(* CODESYS project HomePLC_LinkManager.library
   Company: Tom Oyen
   Description: Link manager
   Version: 1.0
   Placeholder: HomePLC Link Manager
   Author: Tom Oyen
   Title: HomePLC Link Manager

Project tree, tasks and I/O mapping:
  libraries: Tc2_Standard, * (Beckhoff Automation GmbH); Tc2_System, * (Beckhoff Automation GmbH); Tc3_Module, * (Beckhoff Automation GmbH); HomePLC Logging, * (Tom Oyen); HomePLC DIO, * (Tom Oyen)
  POUs/
    IO group/
      DUTs/
        data type E_DIGroupMode
      function block FB_DIGroup [ST]: AddInput, Execute, GetCommand, GetInput, Mode
      function block FB_DOGroup [ST]: AddOutput, Execute, GetOutput, SetCommand
      function block FB_IOGroup [ST]: FB_init, Count
      interface I_DIGroup: AddInput, GetCommand, GetInput, Count, Mode
      interface I_DOGroup: AddOutput, GetOutput, SetCommand, Count
    Link/
      DUTs/
        data type ST_CommandTranslation
      function block FB_Link [ST]: Execute, FB_init, ExcludeFromOverview, InputGroup, OutputGroup, OutputReaction
      interface I_Link: ExcludeFromOverview, InputGroup, OutputGroup, OutputReaction
    function block FB_LinkManager [ST]: CommitLink, Execute, GetLink, Link
    interface I_LinkManager: CommitLink, Link
  Project Information/
    function F_GetCompany [ST]
    function F_GetTitle [ST]
    function F_GetVersion [ST]
  Version/
    global variables Global_Version
*)

// POUs/IO group/DUTs/E_DIGroupMode
{attribute 'qualified_only'}
{attribute 'strict'}
// Mode of combining digital input commands
TYPE E_DIGroupMode :
(
	ModeAND := 0,		// All inputs need to be used to issue the command
	ModeOR	:= 1		// One input is sufficient to issue a command
);
END_TYPE

// POUs/Link/DUTs/ST_CommandTranslation
// Translate input commands to output commands
TYPE ST_CommandTranslation :
STRUCT
	OnShortPress	: E_DOCommand := E_DOCommand.None;	// Output command when input command is short press
	OnLongPress		: E_DOCommand := E_DOCommand.None;	// Output command when input command is long press
	OnDoublePress	: E_DOCommand := E_DOCommand.None;	// Output command when input command is double press
	OnHold			: E_DOCommand := E_DOCommand.None;	// Output command when input command is hold
END_STRUCT
END_TYPE

// Version/Global_Version
{attribute 'TcGenerated'}
{attribute 'no-analysis'}
{attribute 'linkalways'}
// This function has been automatically generated from the project information.
VAR_GLOBAL CONSTANT
	{attribute 'const_non_replaced'}
	stLibVersion_HomePLC_Link_Manager : ST_LibVersion := (iMajor := 1, iMinor := 0, iBuild := 0, iRevision := 0, nFlags := 0, sVersion := '1.0');
END_VAR

// POUs/IO group/FB_DIGroup
// Digital input group
FUNCTION_BLOCK FB_DIGroup EXTENDS FB_IOGroup IMPLEMENTS I_DIGroup
VAR
	aIn				: ARRAY [0..nMaxSize - 1] OF I_DigitalIn;	// Array of interfaces of digital inputs
	eMode			: E_DIGroupMode := E_DIGroupMode.ModeOR;	// Command mode of inputs in group (default = OR)
END_VAR

// Add input to group
METHOD AddInput
VAR_INPUT
	IDI			: I_DigitalIn;
END_VAR
IF nSize < nMaxSize THEN
	aIn[nSize] := IDI;
	nSize := nSize + 1;
END_IF
END_METHOD

// Runs the execute method of all digital input FBs in the group
METHOD Execute
VAR
	i		: INT;
END_VAR
FOR i := 0 TO nSize - 1 DO
	aIn[i].Execute();
END_FOR
END_METHOD

// Determine the command from the inputs in the group
METHOD GetCommand : E_DICommand
VAR
	i				: INT;
	nActive			: INT;
	eCommand		: E_DICommand;
	sTemp			: STRING;
END_VAR
VAR_INST
	eState			: E_DIState;
END_VAR
// Check at least one input is available
IF nSize > 0 THEN
	CASE eMode OF
	E_DIGroupMode.ModeOR:
		// Get command
		eCommand := E_DICommand.None;
		
		FOR i := 0 TO nSize - 1 DO
			// Find first command different from None
			IF aIn[i].Command <> E_DICommand.None THEN
				IF eCommand = E_DICommand.None THEN
					eCommand := aIn[i].Command;
					
					sTemp := 'OR command ';
					sTemp := CONCAT(sTemp, TO_STRING(eCommand));
					fbLogger.AddDebug(sTemp);
				END_IF
			END_IF
		END_FOR
		
		// Issue command
		GetCommand := eCommand;
		
	E_DIGroupMode.ModeAND:
		// Check states
		// Multiple buttons must have been active at the same time with the same state
		nActive := 0;
		FOR i := 0 TO nSize - 1 DO
			IF aIn[i].State <> E_DIState.Idle THEN
				IF eState = E_DIState.Idle THEN
					eState := aIn[i].State;
				END_IF
				IF aIn[i].State = eState THEN
					nActive := nActive + 1;
				END_IF
			END_IF
		END_FOR
		
		// Reset if all inactive
		IF nActive = 0 THEN
			eState := E_DIState.Idle;
		END_IF
		
		// Get command
		eCommand := E_DICommand.None;
		FOR i := 0 TO nSize - 1 DO
			// Find first command different from None
			IF aIn[i].Command <> E_DICommand.None THEN
				IF eCommand = E_DICommand.None THEN
					eCommand := aIn[i].Command;
				END_IF
			END_IF
		END_FOR
		
		IF eCommand <> E_DICommand.None THEN
			// All commands need to be the same
			// Assume command matches detected states
			IF nActive = nSize THEN
				GetCommand := eCommand;
				
				sTemp := 'AND command ';
				sTemp := CONCAT(sTemp, TO_STRING(eCommand));
				sTemp := CONCAT(sTemp, ' by ');
				sTemp := CONCAT(sTemp, INT_TO_STRING(nActive));
				sTemp := CONCAT(sTemp, ' inputs');
				fbLogger.AddDebug(sTemp);
			END_IF
		ELSE
			GetCommand := E_DICommand.None;
		END_IF
	END_CASE
ELSE
	GetCommand := E_DICommand.None;
END_IF
END_METHOD

// Get a specific input from the group
METHOD GetInput : I_DigitalIn
VAR_INPUT
	nInputIndex		: INT;		// Input index
END_VAR
GetInput := aIn[nInputIndex];
END_METHOD

// Set input group mode (default OR)
PROPERTY Mode : E_DIGroupMode
SET
eMode := Mode;
END_SET
END_PROPERTY

END_FUNCTION_BLOCK

// POUs/IO group/FB_IOGroup
{attribute 'reflection'} 
FUNCTION_BLOCK FB_IOGroup
VAR
	nSize			: INT;			// Number of IOs in this group
	
	fbLogger		: class_Tc3EventLogger;
	
	// Use attributes to copy instance name to sName
	{attribute 'instance-path'} 
    {attribute 'noinit'} 
    sName			: STRING; 		// Instance name
END_VAR
VAR CONSTANT
	nMaxSize		: INT := 100;	// Maximum number of IOs in a group
END_VAR

METHOD FB_init : BOOL
VAR_INPUT
	bInitRetains : BOOL; // if TRUE, the retain variables are initialized (warm start / cold start)
	bInCopyCode : BOOL;  // if TRUE, the instance afterwards gets moved into the copy code (online change)
END_VAR
fbLogger.Init(sSource := sName, bEnableVerbose := FALSE);
END_METHOD

// Gets the total number of IOs in the group
PROPERTY Count : INT
GET
Count := nSize;
END_GET
END_PROPERTY

END_FUNCTION_BLOCK

// POUs/IO group/I_DIGroup
INTERFACE I_DIGroup

// Add input to group
METHOD AddInput
VAR_INPUT
	IDI			: I_DigitalIn;		// Digital input
END_VAR
END_METHOD

// Determine the command from the inputs in the group
METHOD GetCommand : E_DICommand
END_METHOD

// Get a specific input from the group
METHOD GetInput : I_DigitalIn
VAR_INPUT
	nInputIndex		: INT;		// Input index
END_VAR
END_METHOD

// Gets the total number of IOs in the group
PROPERTY Count : INT
GET
END_GET
END_PROPERTY

// Set input group mode (default OR)
PROPERTY Mode : E_DIGroupMode
SET
END_SET
END_PROPERTY

END_INTERFACE

// POUs/IO group/FB_DOGroup
// Digital output group
FUNCTION_BLOCK FB_DOGroup EXTENDS FB_IOGroup IMPLEMENTS I_DOGroup
VAR
	aOut		: ARRAY [0..nMaxSize - 1] OF I_DigitalOut;		// Array of interfaces to digital outputs
END_VAR

// Add output to group
METHOD AddOutput
VAR_INPUT
	IDO			: I_DigitalOut;
END_VAR
IF nSize < nMaxSize THEN
	aOut[nSize] := IDO;
	nSize := nSize + 1;
END_IF
END_METHOD

// Runs the execute method of all digital output FBs in the group
METHOD Execute
VAR
	i		: INT;
END_VAR
FOR i := 0 TO nSize - 1 DO
	aOut[i].Execute();
END_FOR
END_METHOD

// Get a specific output from the group
METHOD GetOutput : I_DigitalOut
VAR_INPUT
	nOutputIndex		: INT;		// Output index
END_VAR
GetOutput := aOut[nOutputIndex];
END_METHOD

// Set the command to the outputs in the group
METHOD SetCommand
VAR_INPUT
	eCommand	: E_DOCommand;
END_VAR
VAR
	i			: INT;
END_VAR
FOR i := 0 TO nSize - 1 DO
	IF aOut[i].Command = E_DOCommand.None THEN
		// No command yet, set new command
		aOut[i].SetCommand(eCommand);
	ELSE
		// A command was already issued
		// Do nothing
	END_IF
END_FOR
END_METHOD

END_FUNCTION_BLOCK

// POUs/IO group/I_DOGroup
INTERFACE I_DOGroup

// Add output to group
METHOD AddOutput
VAR_INPUT
	IDO			: I_DigitalOut;		// Digital output
END_VAR
END_METHOD

// Get a specific output from the group
METHOD GetOutput : I_DigitalOut
VAR_INPUT
	nOutputIndex		: INT;		// Output index
END_VAR
END_METHOD

// Set the command to the outputs in the group
METHOD SetCommand
VAR_INPUT
	eCommand	: E_DOCommand;
END_VAR
END_METHOD

// Gets the total number of IOs in the group
PROPERTY Count : INT
GET
END_GET
END_PROPERTY

END_INTERFACE

// POUs/Link/FB_Link
// Link between an input and an output group
FUNCTION_BLOCK FB_Link IMPLEMENTS I_Link
VAR
	IInputGroup				: I_DIGroup;				// Input group interface
	IOutputGroup			: I_DOGroup;				// Output group interface
	
	fbInputGroup			: FB_DIGroup;				// Input group FB, in case interface is not set to an FB
	fbOutputGroup			: FB_DOGroup;				// Output group FB, in case interface is not set to an FB
	
	stCommandTranslation	: ST_CommandTranslation;	// Input command to output command translation
	bExcludeFromOverview	: BOOL;						// Set to true to exclude this link from the links overview
END_VAR

// Execute input group, get its command and then execute the output group with that command
METHOD Execute
// Get input command and translate it to an output command
CASE IInputGroup.GetCommand() OF
	E_DICommand.None:
		IOutputGroup.SetCommand(E_DOCommand.None);
	E_DICommand.ShortPress:
		IOutputGroup.SetCommand(stCommandTranslation.OnShortPress);
	E_DICommand.DoublePress:
		IOutputGroup.SetCommand(stCommandTranslation.OnDoublePress);
	E_DICommand.LongPress:
		IOutputGroup.SetCommand(stCommandTranslation.OnLongPress);
	E_DICommand.Hold:
		IOutputGroup.SetCommand(stCommandTranslation.OnHold);
END_CASE
END_METHOD

METHOD FB_init : BOOL
VAR_INPUT
	bInitRetains : BOOL; // if TRUE, the retain variables are initialized (warm start / cold start)
	bInCopyCode : BOOL;  // if TRUE, the instance afterwards gets moved into the copy code (online change)
END_VAR
// Initialize interfaces with local FBs, can be replaced afterwards if needed
IInputGroup := fbInputGroup;
IOutputGroup := fbOutputGroup;
END_METHOD

// Get/set if the link needs to be excluded from the links overview
PROPERTY ExcludeFromOverview : BOOL
GET
ExcludeFromOverview := bExcludeFromOverview;
END_GET
SET
bExcludeFromOverview := ExcludeFromOverview;
END_SET
END_PROPERTY

// Group of inputs
PROPERTY InputGroup : I_DIGroup
GET
InputGroup := IInputGroup;
END_GET
SET
IInputGroup := InputGroup;
END_SET
END_PROPERTY

// Group of outputs
PROPERTY OutputGroup : I_DOGroup
GET
OutputGroup := IOutputGroup;
END_GET
SET
IOutputGroup := OutputGroup;
END_SET
END_PROPERTY

// Output reaction
PROPERTY OutputReaction : REFERENCE TO ST_CommandTranslation
GET
OutputReaction REF= stCommandTranslation;
END_GET
END_PROPERTY

END_FUNCTION_BLOCK

// POUs/Link/I_Link
INTERFACE I_Link

// Get/set if the link needs to be excluded from the links overview
PROPERTY ExcludeFromOverview : BOOL
GET
END_GET
SET
END_SET
END_PROPERTY

// Group of inputs
PROPERTY InputGroup : I_DIGroup
GET
END_GET
SET
END_SET
END_PROPERTY

// Group of outputs
PROPERTY OutputGroup : I_DOGroup
GET
END_GET
SET
END_SET
END_PROPERTY

// Output reaction
PROPERTY OutputReaction : REFERENCE TO ST_CommandTranslation
GET
END_GET
END_PROPERTY

END_INTERFACE

// POUs/FB_LinkManager
// Link manager
FUNCTION_BLOCK FB_LinkManager IMPLEMENTS I_LinkManager
VAR
	aLinks			: ARRAY [0..nMaxSize - 1] OF FB_Link;	// Array of links
	nSize			: INT;									// Number of links in the array
END_VAR
VAR CONSTANT
	nMaxSize		: INT := 100;							// Maximum number of IOs in a group
END_VAR

// Commit link so it can be executed
METHOD CommitLink
IF nSize < nMaxSize THEN
	nSize := nSize + 1;
END_IF
END_METHOD

// Execute links
METHOD Execute
VAR
	i		: INT;		// Iterator variable
END_VAR
// Execute all links
FOR i := 0 TO nSize - 1 DO
	aLinks[i].Execute();
END_FOR
END_METHOD

METHOD GetLink : I_Link
VAR_INPUT
	nIndex		: INT;		// Link index
END_VAR
GetLink := aLinks[nIndex];
END_METHOD

// Returns a link that can be configured and then committed
PROPERTY Link : I_Link
GET
Link := aLinks[nSize];
END_GET
END_PROPERTY

END_FUNCTION_BLOCK

// POUs/I_LinkManager
// Link manager interface
INTERFACE I_LinkManager

// Commit link so it can be executed
METHOD CommitLink
END_METHOD

// Returns a link that can be configured and then committed
PROPERTY Link : I_Link
GET
END_GET
END_PROPERTY

END_INTERFACE

// Project Information/F_GetCompany
// This function has been automatically generated from the project information.
{attribute 'signature_flag' := '1073741824'}
{attribute 'TcGenerated'}
{attribute 'no-analysis'}
FUNCTION F_GetCompany : WSTRING
VAR_INPUT
	
END_VAR

F_GetCompany := "Tom Oyen";

END_FUNCTION

// Project Information/F_GetTitle
// This function has been automatically generated from the project information.
{attribute 'signature_flag' := '1073741824'}
{attribute 'TcGenerated'}
{attribute 'no-analysis'}
FUNCTION F_GetTitle : WSTRING
VAR_INPUT
	
END_VAR

F_GetTitle := "HomePLC Link Manager";

END_FUNCTION

// Project Information/F_GetVersion
// This function has been automatically generated from the project information.
{attribute 'signature_flag' := '1073741824'}
{attribute 'TcGenerated'}
{attribute 'no-analysis'}
FUNCTION F_GetVersion : ST_LibVersion
VAR_INPUT
	
END_VAR

F_GetVersion.iMajor := 1;
F_GetVersion.iMinor := 0;
F_GetVersion.iBuild := 0;
F_GetVersion.iRevision := 0;
F_GetVersion.sVersion := '1.0';
F_GetVersion.nFlags := 0;

END_FUNCTION
